(* Logix 5000 project; controller SX_V040001_C001 vendor 1 type 14 code 77 rev 16.22; software revision 16.04; part 12 of 35 *)
(* tags used below, declared in another part *)
   ALL_KINDS : INT[90];
   C_MINUTES : COUNTER;
   C_SECONDS : COUNTER;
   CMD : INT[36];
   DRIVE : INT[32];
   EMPTYING : INT[18];
   G_DInput : DINT[3];
   G_DOutput : DINT[3];
   loading : INT[19];
   louvre : INT[11];
   m_alarm_exist : BOOL;
   m_alarm_horn : BOOL;
   m_battery_low : BOOL;
   m_on_off_line : BOOL;
   m_power_up : BOOL;
   METERING : INT[44];
   PARAMETER : INT[501];
   RM_CMD : INT[9];
   STATUS_GENERAL : INT[135];
   TEMP : INT[14];
(* MainProgram, continued *)

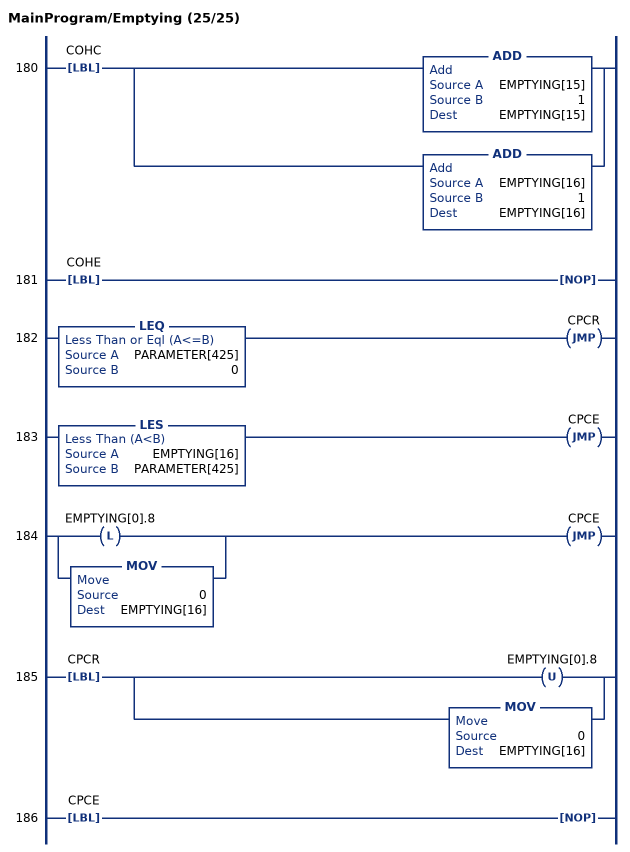
   [picture p260: MainProgram/Emptying rungs 180-186]
   180: LBL(COHC)[ADD(EMPTYING[15],1,EMPTYING[15]) ,ADD(EMPTYING[16],1,EMPTYING[16]) ];
   181: LBL(COHE)NOP();
   182: LEQ(PARAMETER[425],0)JMP(CPCR);
   183: LES(EMPTYING[16],PARAMETER[425])JMP(CPCE);
   184: [OTL(EMPTYING[0].8) ,MOV(0,EMPTYING[16]) ]JMP(CPCE);
   185: LBL(CPCR)[OTU(EMPTYING[0].8) ,MOV(0,EMPTYING[16]) ];
   186: LBL(CPCE)NOP();
END_ROUTINE

ROUTINE FirstScan   (* ladder *)
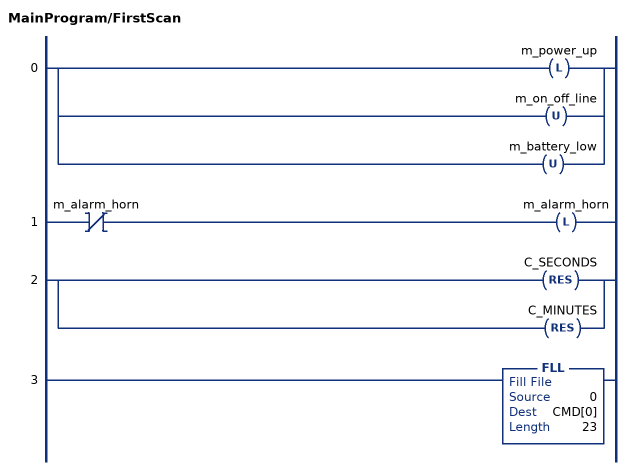
   0: [OTL(m_power_up) ,OTU(m_on_off_line) ,OTU(m_battery_low) ];
   1: XIO(m_alarm_horn)OTL(m_alarm_horn);
   2: [RES(C_SECONDS) ,RES(C_MINUTES) ];
   3: FLL(0,CMD[0],23);
END_ROUTINE

ROUTINE GenerateStatus   (* ladder *)
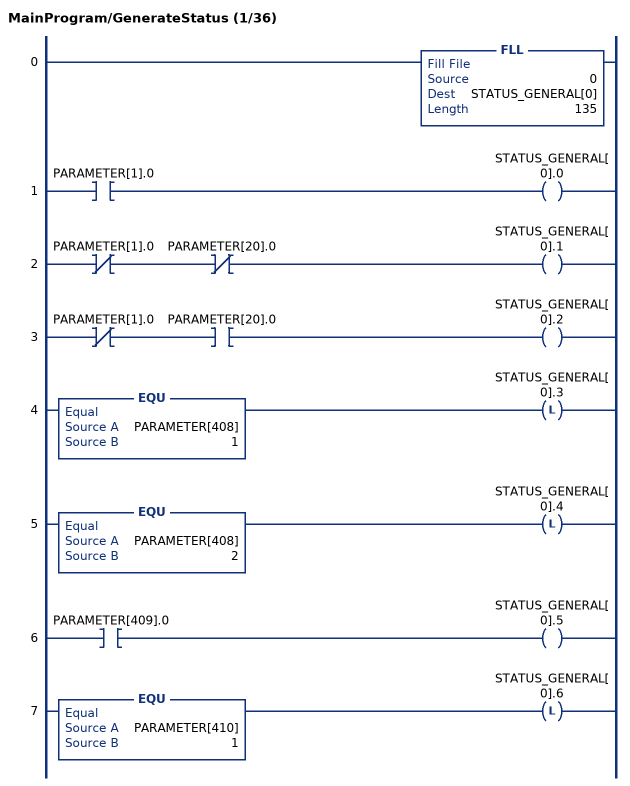
   0: FLL(0,STATUS_GENERAL[0],135);
   1: XIC(PARAMETER[1].0)OTE(STATUS_GENERAL[0].0);
   2: XIO(PARAMETER[1].0)XIO(PARAMETER[20].0)OTE(STATUS_GENERAL[0].1);
   3: XIO(PARAMETER[1].0)XIC(PARAMETER[20].0)OTE(STATUS_GENERAL[0].2);
   4: EQU(PARAMETER[408],1)OTL(STATUS_GENERAL[0].3);
   5: EQU(PARAMETER[408],2)OTL(STATUS_GENERAL[0].4);
   6: XIC(PARAMETER[409].0)OTE(STATUS_GENERAL[0].5);
   7: EQU(PARAMETER[410],1)OTL(STATUS_GENERAL[0].6);
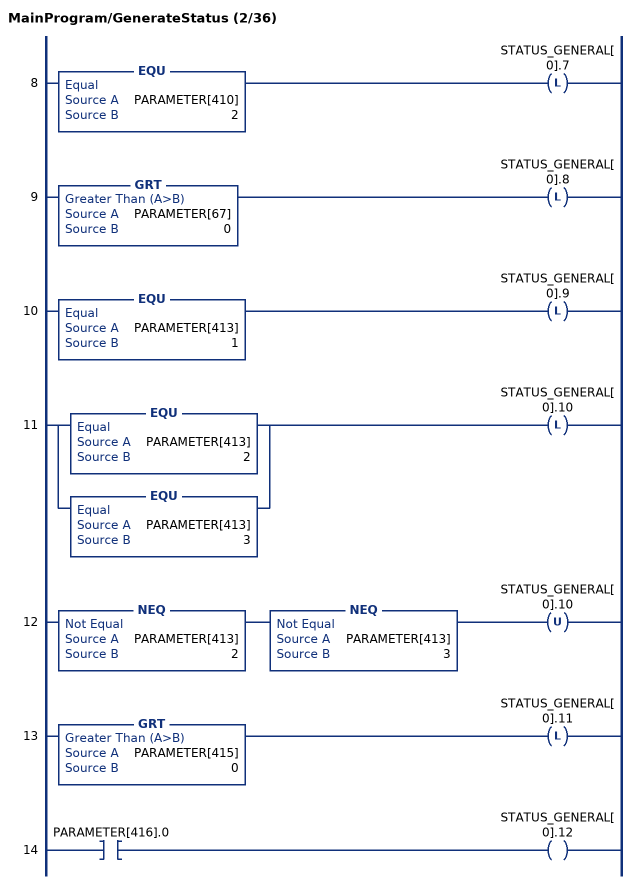
   8: EQU(PARAMETER[410],2)OTL(STATUS_GENERAL[0].7);
   9: GRT(PARAMETER[67],0)OTL(STATUS_GENERAL[0].8);
   10: EQU(PARAMETER[413],1)OTL(STATUS_GENERAL[0].9);
   11: [EQU(PARAMETER[413],2) ,EQU(PARAMETER[413],3) ]OTL(STATUS_GENERAL[0].10);
   12: NEQ(PARAMETER[413],2)NEQ(PARAMETER[413],3)OTU(STATUS_GENERAL[0].10);
   13: GRT(PARAMETER[415],0)OTL(STATUS_GENERAL[0].11);
   14: XIC(PARAMETER[416].0)OTE(STATUS_GENERAL[0].12);
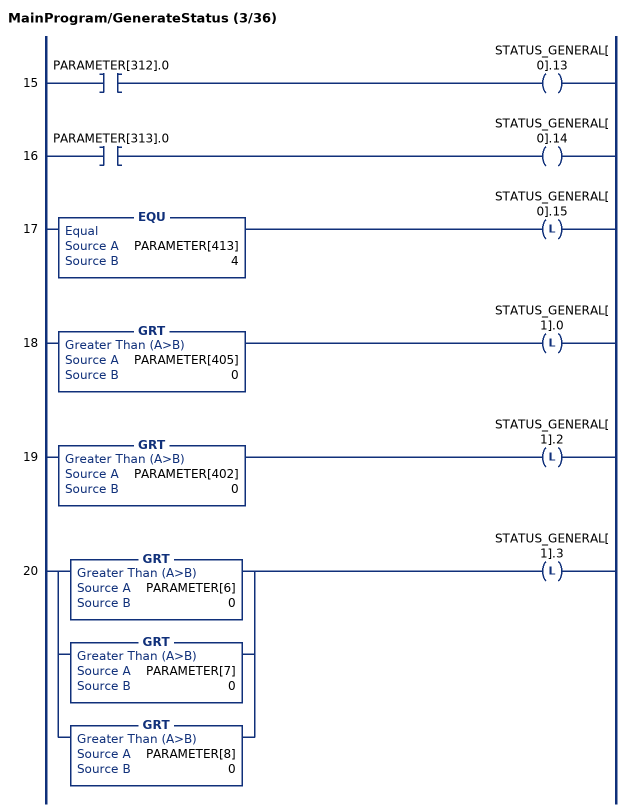
   15: XIC(PARAMETER[312].0)OTE(STATUS_GENERAL[0].13);
   16: XIC(PARAMETER[313].0)OTE(STATUS_GENERAL[0].14);
   17: EQU(PARAMETER[413],4)OTL(STATUS_GENERAL[0].15);
   18: GRT(PARAMETER[405],0)OTL(STATUS_GENERAL[1].0);
   19: GRT(PARAMETER[402],0)OTL(STATUS_GENERAL[1].2);
   20: [GRT(PARAMETER[6],0) ,GRT(PARAMETER[7],0) ,GRT(PARAMETER[8],0) ]OTL(STATUS_GENERAL[1].3);
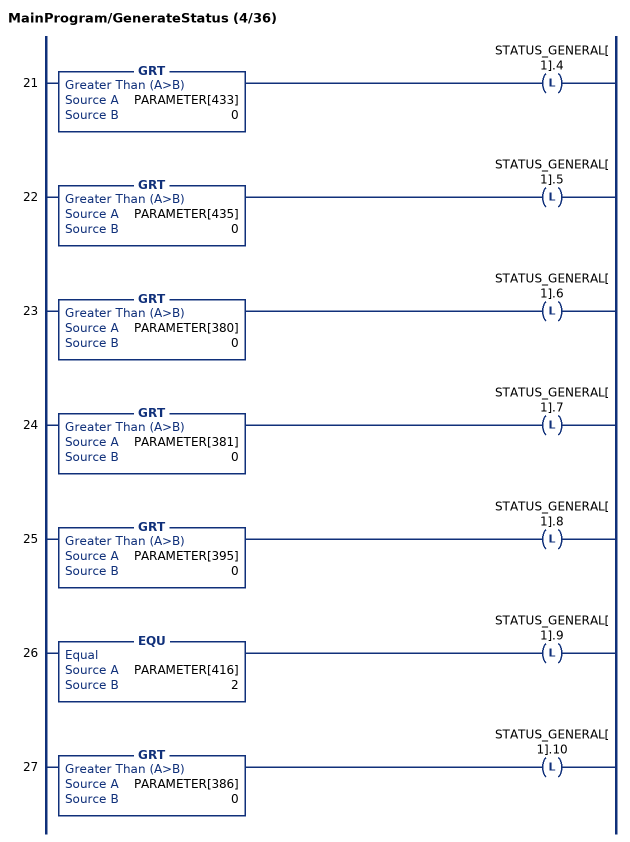
   21: GRT(PARAMETER[433],0)OTL(STATUS_GENERAL[1].4);
   22: GRT(PARAMETER[435],0)OTL(STATUS_GENERAL[1].5);
   23: GRT(PARAMETER[380],0)OTL(STATUS_GENERAL[1].6);
   24: GRT(PARAMETER[381],0)OTL(STATUS_GENERAL[1].7);
   25: GRT(PARAMETER[395],0)OTL(STATUS_GENERAL[1].8);
   26: EQU(PARAMETER[416],2)OTL(STATUS_GENERAL[1].9);
   27: GRT(PARAMETER[386],0)OTL(STATUS_GENERAL[1].10);
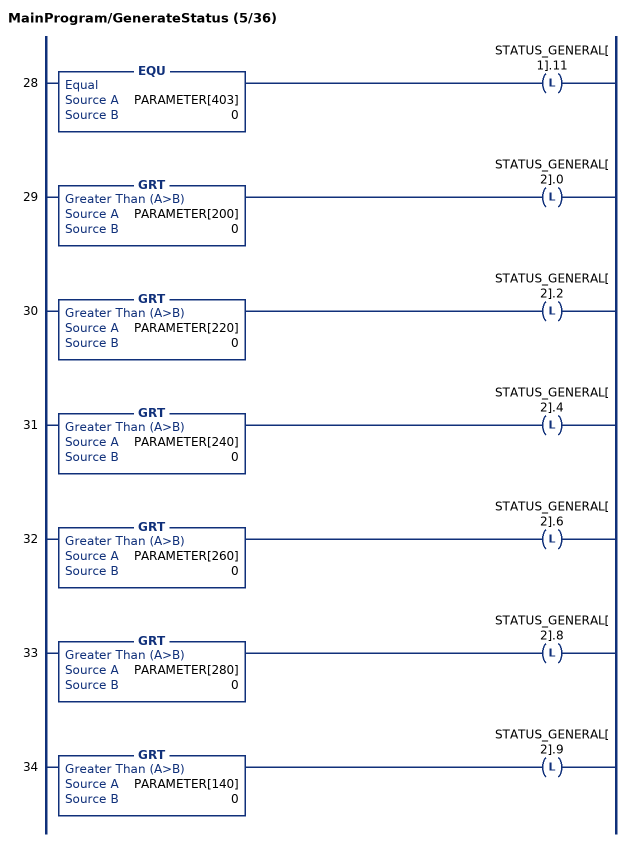
   28: EQU(PARAMETER[403],0)OTL(STATUS_GENERAL[1].11);
   29: GRT(PARAMETER[200],0)OTL(STATUS_GENERAL[2].0);
   30: GRT(PARAMETER[220],0)OTL(STATUS_GENERAL[2].2);
   31: GRT(PARAMETER[240],0)OTL(STATUS_GENERAL[2].4);
   32: GRT(PARAMETER[260],0)OTL(STATUS_GENERAL[2].6);
   33: GRT(PARAMETER[280],0)OTL(STATUS_GENERAL[2].8);
   34: GRT(PARAMETER[140],0)OTL(STATUS_GENERAL[2].9);
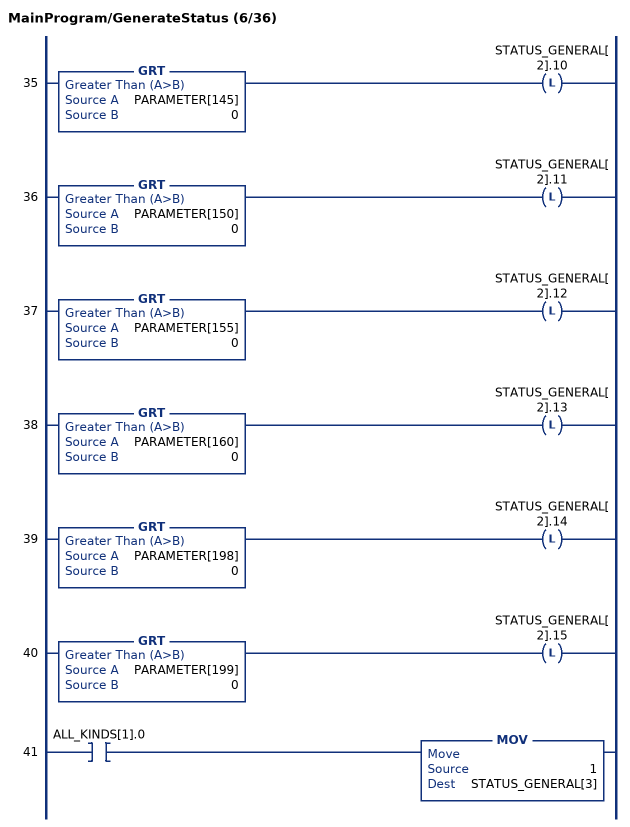
   35: GRT(PARAMETER[145],0)OTL(STATUS_GENERAL[2].10);
   36: GRT(PARAMETER[150],0)OTL(STATUS_GENERAL[2].11);
   37: GRT(PARAMETER[155],0)OTL(STATUS_GENERAL[2].12);
   38: GRT(PARAMETER[160],0)OTL(STATUS_GENERAL[2].13);
   39: GRT(PARAMETER[198],0)OTL(STATUS_GENERAL[2].14);
   40: GRT(PARAMETER[199],0)OTL(STATUS_GENERAL[2].15);
   41: XIC(ALL_KINDS[1].0)MOV(1,STATUS_GENERAL[3]);
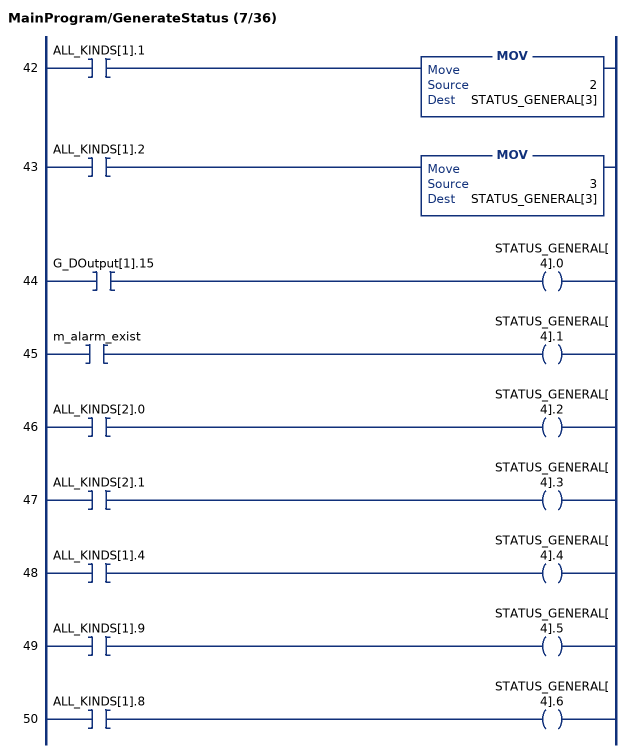
   42: XIC(ALL_KINDS[1].1)MOV(2,STATUS_GENERAL[3]);
   43: XIC(ALL_KINDS[1].2)MOV(3,STATUS_GENERAL[3]);
   44: XIC(G_DOutput[1].15)OTE(STATUS_GENERAL[4].0);
   45: XIC(m_alarm_exist)OTE(STATUS_GENERAL[4].1);
   46: XIC(ALL_KINDS[2].0)OTE(STATUS_GENERAL[4].2);
   47: XIC(ALL_KINDS[2].1)OTE(STATUS_GENERAL[4].3);
   48: XIC(ALL_KINDS[1].4)OTE(STATUS_GENERAL[4].4);
   49: XIC(ALL_KINDS[1].9)OTE(STATUS_GENERAL[4].5);
   50: XIC(ALL_KINDS[1].8)OTE(STATUS_GENERAL[4].6);
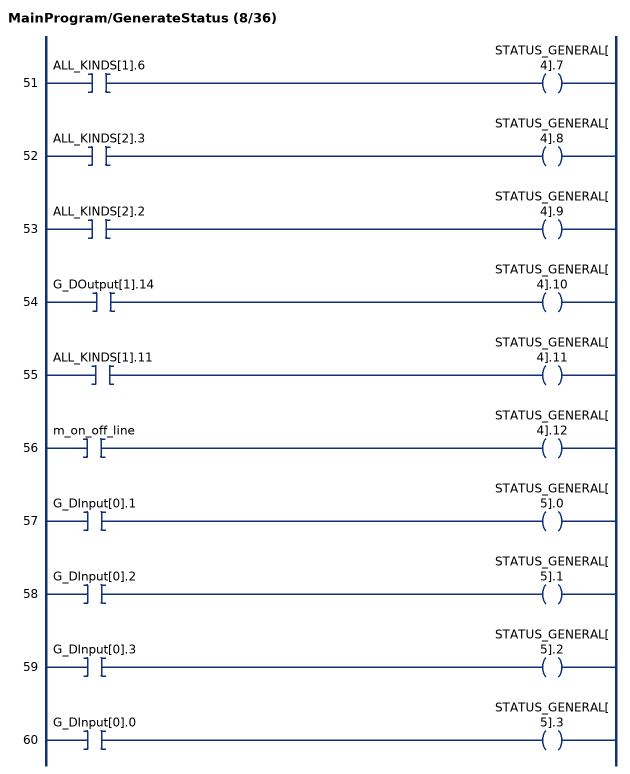
   51: XIC(ALL_KINDS[1].6)OTE(STATUS_GENERAL[4].7);
   52: XIC(ALL_KINDS[2].3)OTE(STATUS_GENERAL[4].8);
   53: XIC(ALL_KINDS[2].2)OTE(STATUS_GENERAL[4].9);
   54: XIC(G_DOutput[1].14)OTE(STATUS_GENERAL[4].10);
   55: XIC(ALL_KINDS[1].11)OTE(STATUS_GENERAL[4].11);
   56: XIC(m_on_off_line)OTE(STATUS_GENERAL[4].12);
   57: XIC(G_DInput[0].1)OTE(STATUS_GENERAL[5].0);
   58: XIC(G_DInput[0].2)OTE(STATUS_GENERAL[5].1);
   59: XIC(G_DInput[0].3)OTE(STATUS_GENERAL[5].2);
   60: XIC(G_DInput[0].0)OTE(STATUS_GENERAL[5].3);
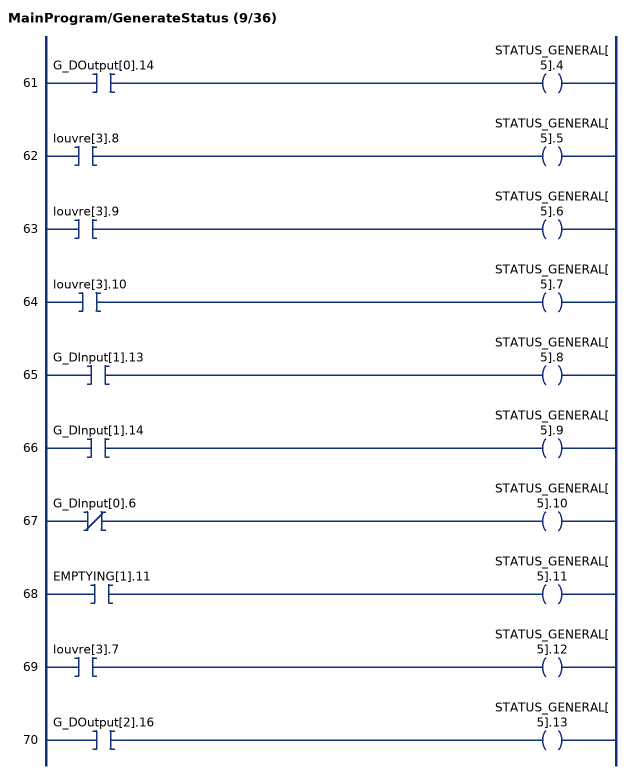
   61: XIC(G_DOutput[0].14)OTE(STATUS_GENERAL[5].4);
   62: XIC(louvre[3].8)OTE(STATUS_GENERAL[5].5);
   63: XIC(louvre[3].9)OTE(STATUS_GENERAL[5].6);
   64: XIC(louvre[3].10)OTE(STATUS_GENERAL[5].7);
   65: XIC(G_DInput[1].13)OTE(STATUS_GENERAL[5].8);
   66: XIC(G_DInput[1].14)OTE(STATUS_GENERAL[5].9);
   67: XIO(G_DInput[0].6)OTE(STATUS_GENERAL[5].10);
   68: XIC(EMPTYING[1].11)OTE(STATUS_GENERAL[5].11);
   69: XIC(louvre[3].7)OTE(STATUS_GENERAL[5].12);
   70: XIC(G_DOutput[2].16)OTE(STATUS_GENERAL[5].13);
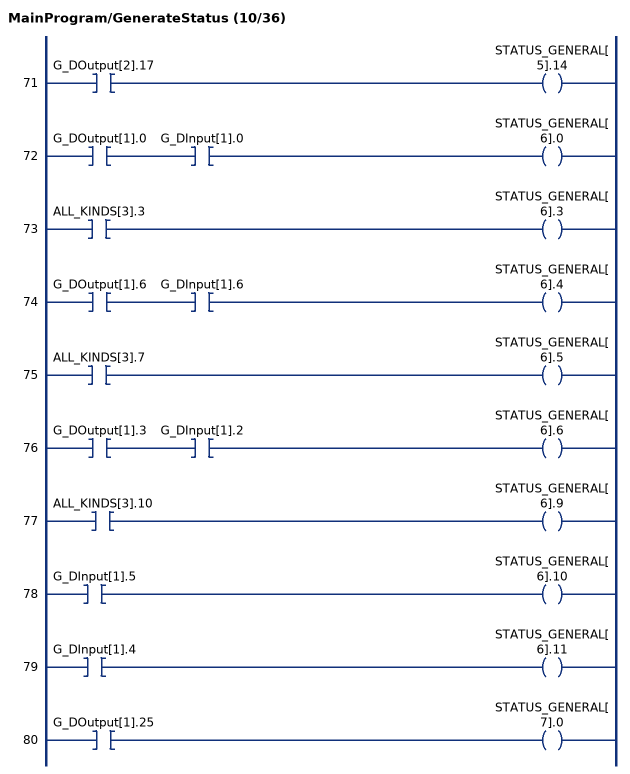
   71: XIC(G_DOutput[2].17)OTE(STATUS_GENERAL[5].14);
   72: XIC(G_DOutput[1].0)XIC(G_DInput[1].0)OTE(STATUS_GENERAL[6].0);
   73: XIC(ALL_KINDS[3].3)OTE(STATUS_GENERAL[6].3);
   74: XIC(G_DOutput[1].6)XIC(G_DInput[1].6)OTE(STATUS_GENERAL[6].4);
   75: XIC(ALL_KINDS[3].7)OTE(STATUS_GENERAL[6].5);
   76: XIC(G_DOutput[1].3)XIC(G_DInput[1].2)OTE(STATUS_GENERAL[6].6);
   77: XIC(ALL_KINDS[3].10)OTE(STATUS_GENERAL[6].9);
   78: XIC(G_DInput[1].5)OTE(STATUS_GENERAL[6].10);
   79: XIC(G_DInput[1].4)OTE(STATUS_GENERAL[6].11);
   80: XIC(G_DOutput[1].25)OTE(STATUS_GENERAL[7].0);
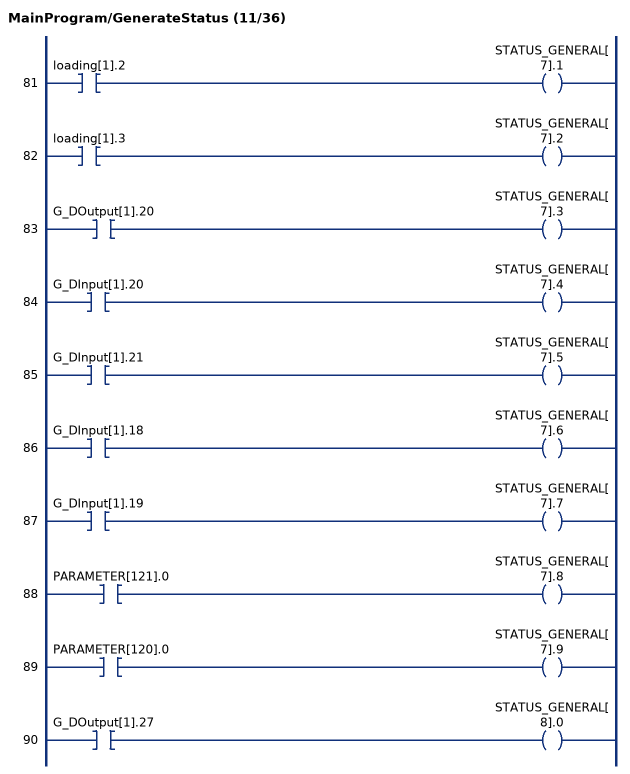
   81: XIC(loading[1].2)OTE(STATUS_GENERAL[7].1);
   82: XIC(loading[1].3)OTE(STATUS_GENERAL[7].2);
   83: XIC(G_DOutput[1].20)OTE(STATUS_GENERAL[7].3);
   84: XIC(G_DInput[1].20)OTE(STATUS_GENERAL[7].4);
   85: XIC(G_DInput[1].21)OTE(STATUS_GENERAL[7].5);
   86: XIC(G_DInput[1].18)OTE(STATUS_GENERAL[7].6);
   87: XIC(G_DInput[1].19)OTE(STATUS_GENERAL[7].7);
   88: XIC(PARAMETER[121].0)OTE(STATUS_GENERAL[7].8);
   89: XIC(PARAMETER[120].0)OTE(STATUS_GENERAL[7].9);
   90: XIC(G_DOutput[1].27)OTE(STATUS_GENERAL[8].0);
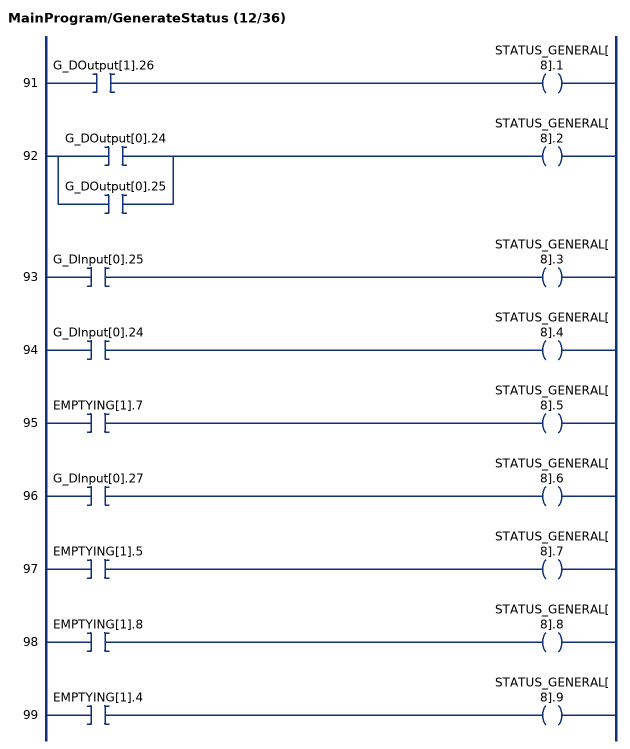
   91: XIC(G_DOutput[1].26)OTE(STATUS_GENERAL[8].1);
   92: [XIC(G_DOutput[0].24) ,XIC(G_DOutput[0].25) ]OTE(STATUS_GENERAL[8].2);
   93: XIC(G_DInput[0].25)OTE(STATUS_GENERAL[8].3);
   94: XIC(G_DInput[0].24)OTE(STATUS_GENERAL[8].4);
   95: XIC(EMPTYING[1].7)OTE(STATUS_GENERAL[8].5);
   96: XIC(G_DInput[0].27)OTE(STATUS_GENERAL[8].6);
   97: XIC(EMPTYING[1].5)OTE(STATUS_GENERAL[8].7);
   98: XIC(EMPTYING[1].8)OTE(STATUS_GENERAL[8].8);
   99: XIC(EMPTYING[1].4)OTE(STATUS_GENERAL[8].9);
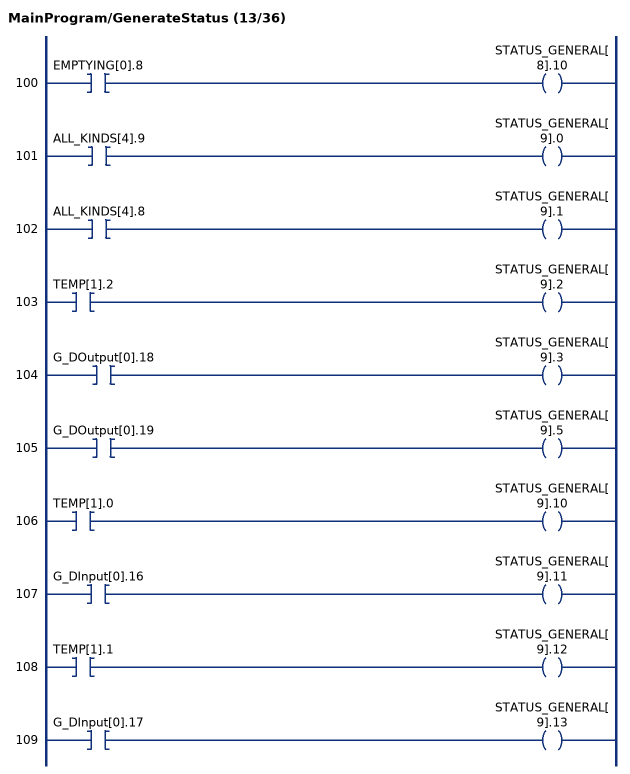
   100: XIC(EMPTYING[0].8)OTE(STATUS_GENERAL[8].10);
   101: XIC(ALL_KINDS[4].9)OTE(STATUS_GENERAL[9].0);
   102: XIC(ALL_KINDS[4].8)OTE(STATUS_GENERAL[9].1);
   103: XIC(TEMP[1].2)OTE(STATUS_GENERAL[9].2);
   104: XIC(G_DOutput[0].18)OTE(STATUS_GENERAL[9].3);
   105: XIC(G_DOutput[0].19)OTE(STATUS_GENERAL[9].5);
   106: XIC(TEMP[1].0)OTE(STATUS_GENERAL[9].10);
   107: XIC(G_DInput[0].16)OTE(STATUS_GENERAL[9].11);
   108: XIC(TEMP[1].1)OTE(STATUS_GENERAL[9].12);
   109: XIC(G_DInput[0].17)OTE(STATUS_GENERAL[9].13);
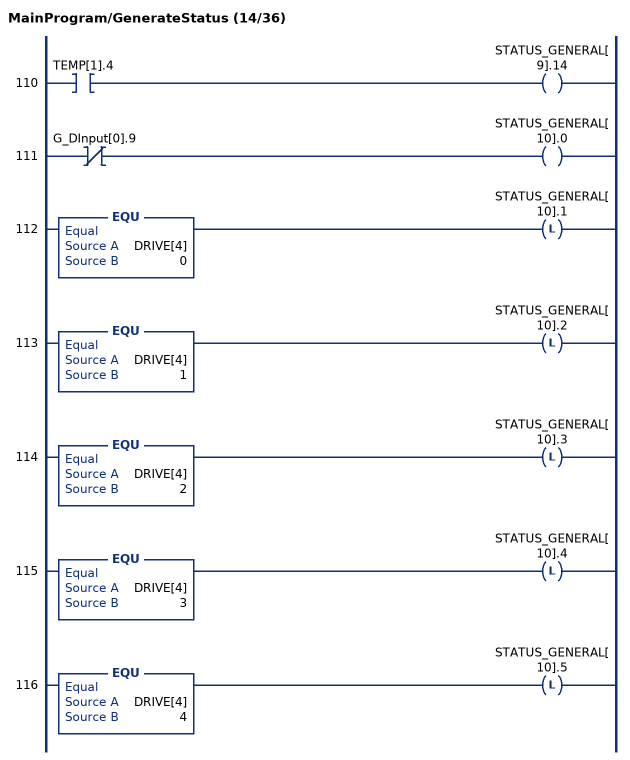
   110: XIC(TEMP[1].4)OTE(STATUS_GENERAL[9].14);
   111: XIO(G_DInput[0].9)OTE(STATUS_GENERAL[10].0);
   112: EQU(DRIVE[4],0)OTL(STATUS_GENERAL[10].1);
   113: EQU(DRIVE[4],1)OTL(STATUS_GENERAL[10].2);
   114: EQU(DRIVE[4],2)OTL(STATUS_GENERAL[10].3);
   115: EQU(DRIVE[4],3)OTL(STATUS_GENERAL[10].4);
   116: EQU(DRIVE[4],4)OTL(STATUS_GENERAL[10].5);
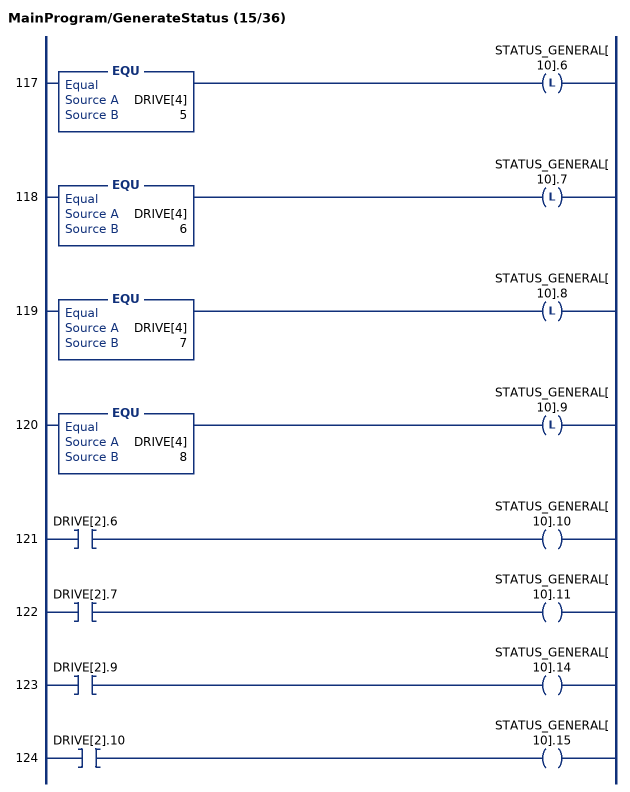
   117: EQU(DRIVE[4],5)OTL(STATUS_GENERAL[10].6);
   118: EQU(DRIVE[4],6)OTL(STATUS_GENERAL[10].7);
   119: EQU(DRIVE[4],7)OTL(STATUS_GENERAL[10].8);
   120: EQU(DRIVE[4],8)OTL(STATUS_GENERAL[10].9);
   121: XIC(DRIVE[2].6)OTE(STATUS_GENERAL[10].10);
   122: XIC(DRIVE[2].7)OTE(STATUS_GENERAL[10].11);
   123: XIC(DRIVE[2].9)OTE(STATUS_GENERAL[10].14);
   124: XIC(DRIVE[2].10)OTE(STATUS_GENERAL[10].15);
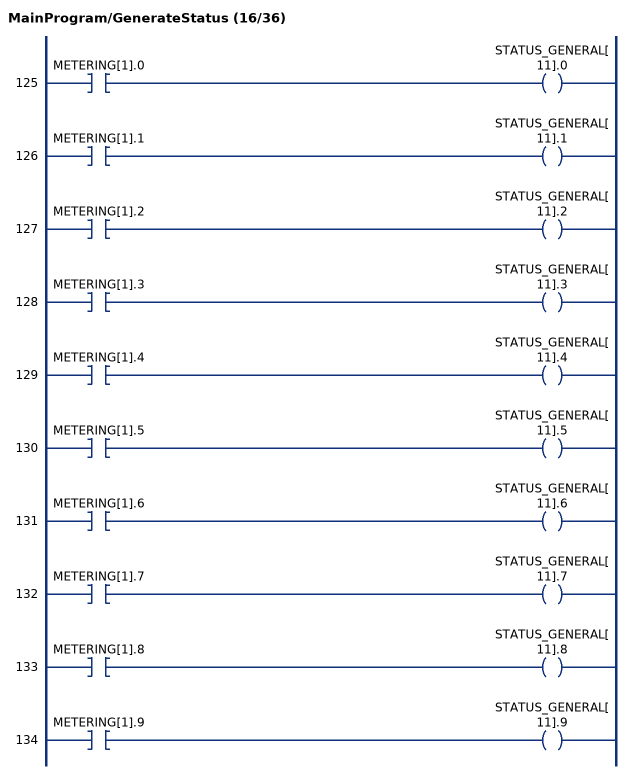
   125: XIC(METERING[1].0)OTE(STATUS_GENERAL[11].0);
   126: XIC(METERING[1].1)OTE(STATUS_GENERAL[11].1);
   127: XIC(METERING[1].2)OTE(STATUS_GENERAL[11].2);
   128: XIC(METERING[1].3)OTE(STATUS_GENERAL[11].3);
   129: XIC(METERING[1].4)OTE(STATUS_GENERAL[11].4);
   130: XIC(METERING[1].5)OTE(STATUS_GENERAL[11].5);
   131: XIC(METERING[1].6)OTE(STATUS_GENERAL[11].6);
   132: XIC(METERING[1].7)OTE(STATUS_GENERAL[11].7);
   133: XIC(METERING[1].8)OTE(STATUS_GENERAL[11].8);
   134: XIC(METERING[1].9)OTE(STATUS_GENERAL[11].9);
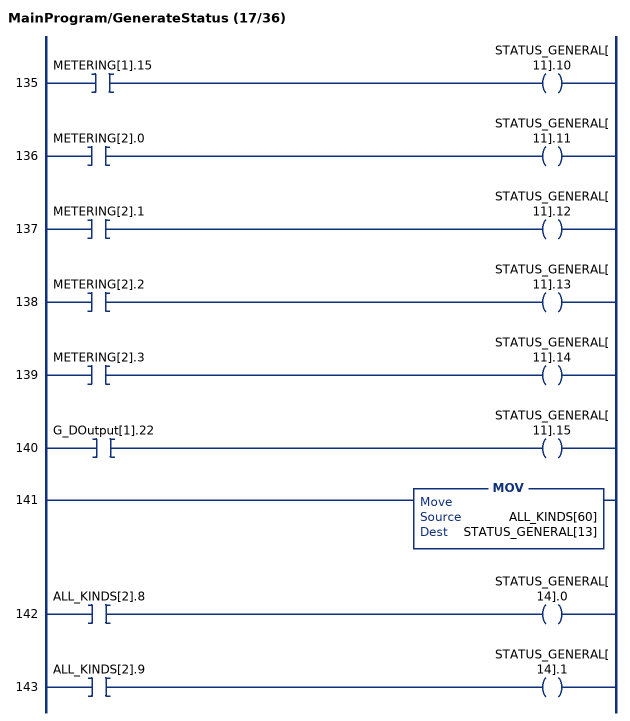
   135: XIC(METERING[1].15)OTE(STATUS_GENERAL[11].10);
   136: XIC(METERING[2].0)OTE(STATUS_GENERAL[11].11);
   137: XIC(METERING[2].1)OTE(STATUS_GENERAL[11].12);
   138: XIC(METERING[2].2)OTE(STATUS_GENERAL[11].13);
   139: XIC(METERING[2].3)OTE(STATUS_GENERAL[11].14);
   140: XIC(G_DOutput[1].22)OTE(STATUS_GENERAL[11].15);
   141: MOV(ALL_KINDS[60],STATUS_GENERAL[13]);
   142: XIC(ALL_KINDS[2].8)OTE(STATUS_GENERAL[14].0);
   143: XIC(ALL_KINDS[2].9)OTE(STATUS_GENERAL[14].1);
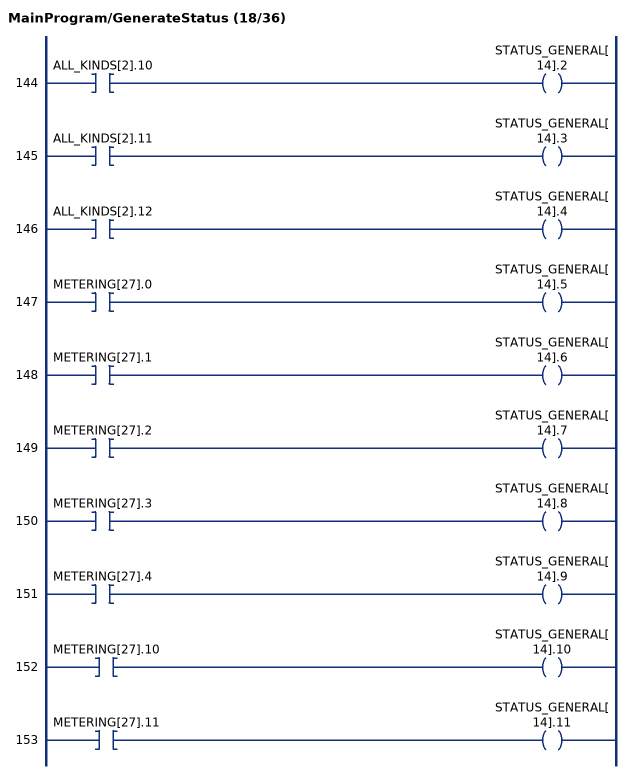
   144: XIC(ALL_KINDS[2].10)OTE(STATUS_GENERAL[14].2);
   145: XIC(ALL_KINDS[2].11)OTE(STATUS_GENERAL[14].3);
   146: XIC(ALL_KINDS[2].12)OTE(STATUS_GENERAL[14].4);
   147: XIC(METERING[27].0)OTE(STATUS_GENERAL[14].5);
   148: XIC(METERING[27].1)OTE(STATUS_GENERAL[14].6);
   149: XIC(METERING[27].2)OTE(STATUS_GENERAL[14].7);
   150: XIC(METERING[27].3)OTE(STATUS_GENERAL[14].8);
   151: XIC(METERING[27].4)OTE(STATUS_GENERAL[14].9);
   152: XIC(METERING[27].10)OTE(STATUS_GENERAL[14].10);
   153: XIC(METERING[27].11)OTE(STATUS_GENERAL[14].11);
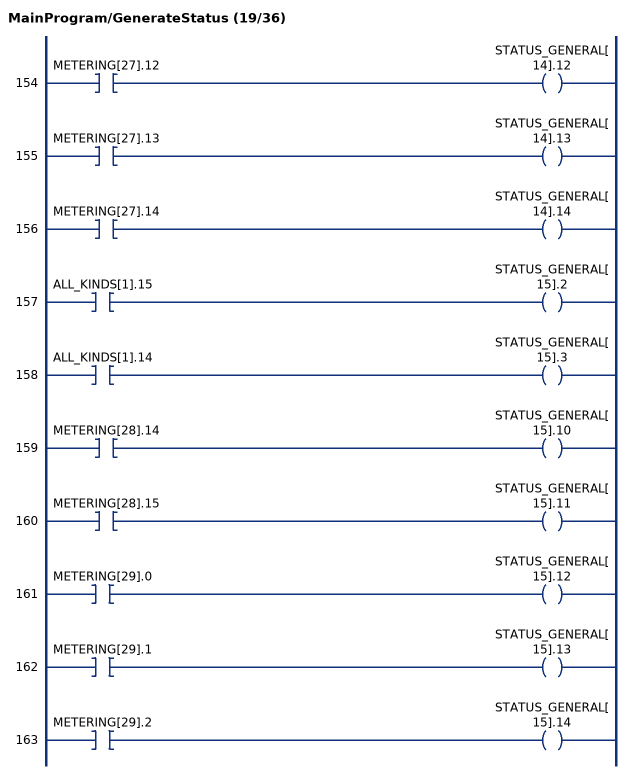
   154: XIC(METERING[27].12)OTE(STATUS_GENERAL[14].12);
   155: XIC(METERING[27].13)OTE(STATUS_GENERAL[14].13);
   156: XIC(METERING[27].14)OTE(STATUS_GENERAL[14].14);
   157: XIC(ALL_KINDS[1].15)OTE(STATUS_GENERAL[15].2);
   158: XIC(ALL_KINDS[1].14)OTE(STATUS_GENERAL[15].3);
   159: XIC(METERING[28].14)OTE(STATUS_GENERAL[15].10);
   160: XIC(METERING[28].15)OTE(STATUS_GENERAL[15].11);
   161: XIC(METERING[29].0)OTE(STATUS_GENERAL[15].12);
   162: XIC(METERING[29].1)OTE(STATUS_GENERAL[15].13);
   163: XIC(METERING[29].2)OTE(STATUS_GENERAL[15].14);
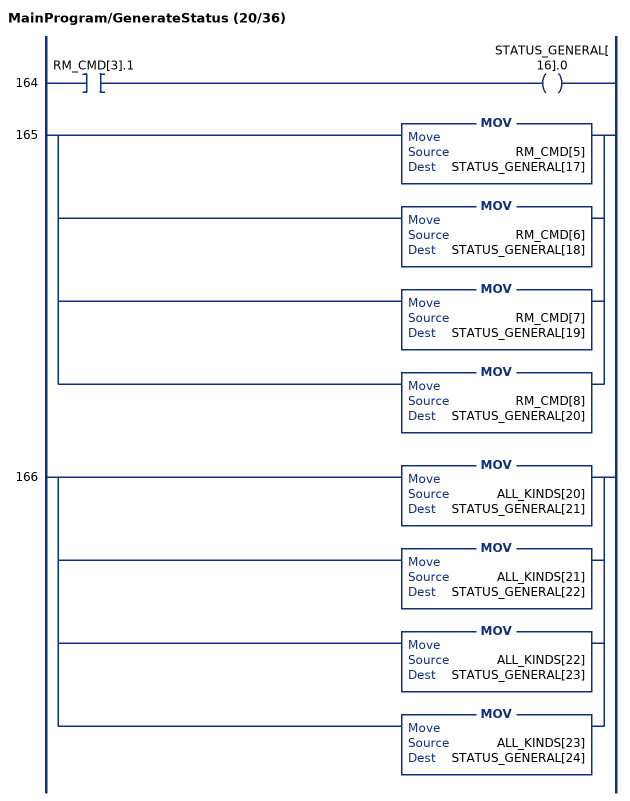
   164: XIC(RM_CMD[3].1)OTE(STATUS_GENERAL[16].0);
   165: [MOV(RM_CMD[5],STATUS_GENERAL[17]) ,MOV(RM_CMD[6],STATUS_GENERAL[18]) ,MOV(RM_CMD[7],STATUS_GENERAL[19]) ,MOV(RM_CMD[8],STATUS_GENERAL[20]) ];
   166: [MOV(ALL_KINDS[20],STATUS_GENERAL[21]) ,MOV(ALL_KINDS[21],STATUS_GENERAL[22]) ,MOV(ALL_KINDS[22],STATUS_GENERAL[23]) ,MOV(ALL_KINDS[23],STATUS_GENERAL[24]) ];
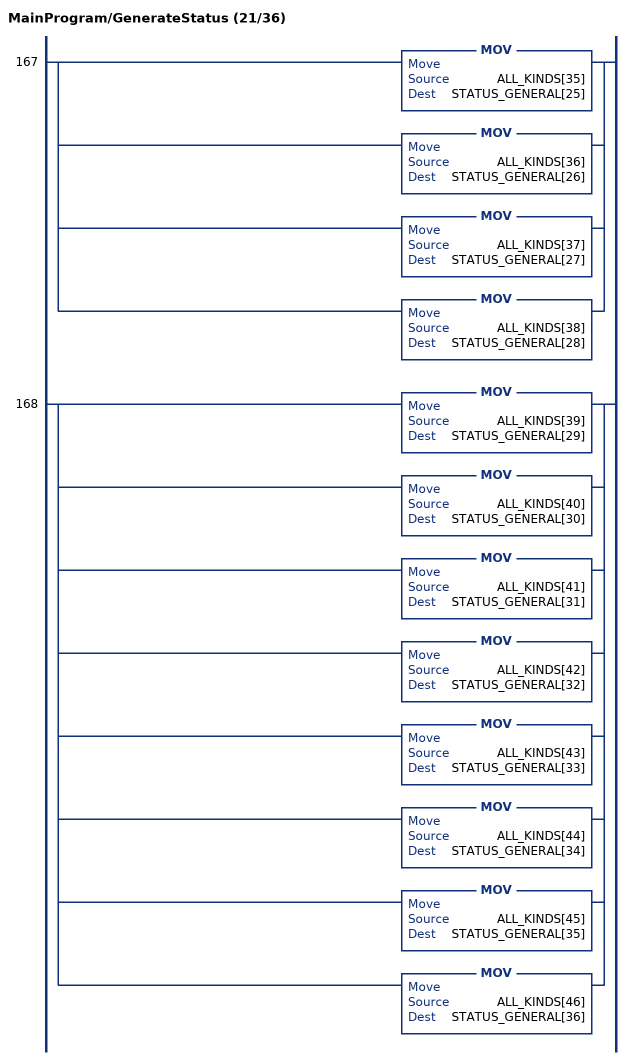
   167: [MOV(ALL_KINDS[35],STATUS_GENERAL[25]) ,MOV(ALL_KINDS[36],STATUS_GENERAL[26]) ,MOV(ALL_KINDS[37],STATUS_GENERAL[27]) ,MOV(ALL_KINDS[38],STATUS_GENERAL[28]) ];
   168: [MOV(ALL_KINDS[39],STATUS_GENERAL[29]) ,MOV(ALL_KINDS[40],STATUS_GENERAL[30]) ,MOV(ALL_KINDS[41],STATUS_GENERAL[31]) ,MOV(ALL_KINDS[42],STATUS_GENERAL[32]) ,MOV(ALL_KINDS[43],STATUS_GENERAL[33]) ,MOV(ALL_KINDS[44],STATUS_GENERAL[34]) ,MOV(ALL_KINDS[45],STATUS_GENERAL[35]) ,MOV(ALL_KINDS[46],STATUS_GENERAL[36]) ];
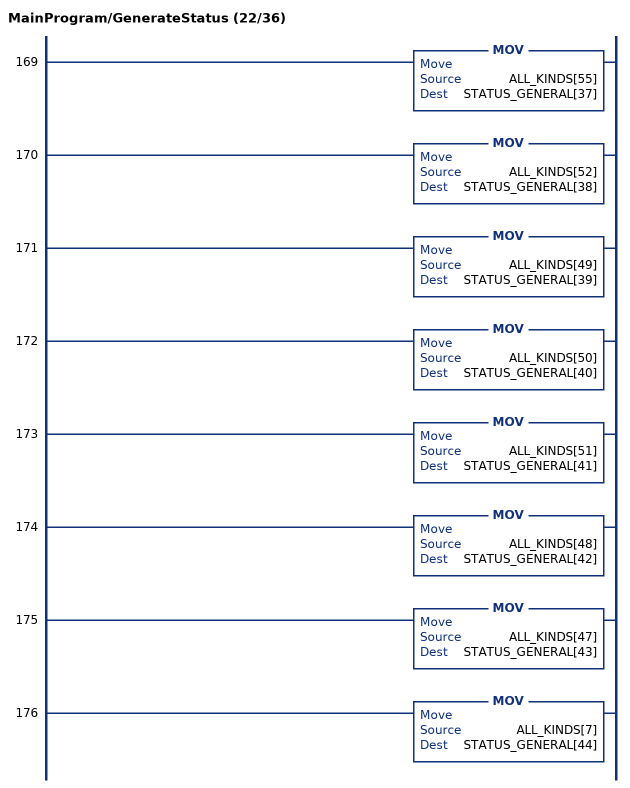
   169: MOV(ALL_KINDS[55],STATUS_GENERAL[37]);
   170: MOV(ALL_KINDS[52],STATUS_GENERAL[38]);
   171: MOV(ALL_KINDS[49],STATUS_GENERAL[39]);
   172: MOV(ALL_KINDS[50],STATUS_GENERAL[40]);
   173: MOV(ALL_KINDS[51],STATUS_GENERAL[41]);
   174: MOV(ALL_KINDS[48],STATUS_GENERAL[42]);
   175: MOV(ALL_KINDS[47],STATUS_GENERAL[43]);
   176: MOV(ALL_KINDS[7],STATUS_GENERAL[44]);
